//==================================================================================================
//							Beckhoff Automation Poland
//									18.05.2018
//	Struktura interfejsu do obslugi Axis Online
//	v1.1	|| TC v 3.1.4022.16		|| - zmiana nazw struktur 
// 									 ST_FBCoEAX8000SetPositionOffsetIO 	--> ST_FBCoESetPositionOffsetIO
// 									 ST_FBHoldingBrakeCtrlAX8000IO 		--> ST_FBHoldingBrakeCtrlIO
// 									 ST_FBMotorMonitoringAX8000IO 		--> ST_FBMotorMonitoringIO
//  v1.0	|| TC v 3.1.4022.16		|| - pierwsza wersja
//==================================================================================================
TYPE ST_McAxisOnline :
STRUCT
	// Base administration
	mcPower							: ST_MCPowerIO;
	mcStop							: ST_MCStopIO;
	mcHalt							: ST_MCHaltIO;
	mcSS1							: ST_MCStopIO;
	mcSS2							: ST_MCStopIO;
	mcReset							: ST_MCResetIO;
	mcHome							: ST_MCHomeIO;
	mcSetPosition					: ST_MCSetPositionIO;
	stSetPositionOffset				: ST_FBSetPositionOffsetIO;
	// Base move
	mcMoveAbsolute					: ST_MCMoveAbsoluteIO;
	mcMoveRelative					: ST_MCMoveRelativeIO;
	mcMoveVelocity					: ST_MCMoveVelocityIO;
	mcMoveModulo					: ST_MCMoveModuloIO;
	mcMoveAbsolute2					: ST_MCMoveAbsoluteIO;
	mcMoveRelative2					: ST_MCMoveRelativeIO;
	mcMoveVelocity2					: ST_MCMoveVelocityIO;
	mcMoveModulo2					: ST_MCMoveModuloIO;
	mcJog							: ST_MCJogIO;
	// States, parameters, monitoring and diag
	stMotorMonitoring				: ST_FBMotorMonitoringIO;
	stHoldingBrake					: ST_FBHoldingBrakeCtrlIO;
	stNcLimitSwitch					: ST_FBNcSWLimitSwitchCtrlIO;
	stAxisParameter					: Tc2_MC2.ST_AxisParameterSet;
	stDriveRef						: Tc2_EtherCAT.ST_DriveRef;
	stDriveAddress					: Tc2_MC2.ST_DriveAddress;
	stChannelErrorCode				: ST_FBReadChannelErrorCodeIO;
	stStatus						: ST_McAxisStatus;
	// FBs
	stGetDriveRef					: ST_FBGetDriveRefIO;					// IO for FB_GetDriveRef
	mcReadDriveAddress				: ST_MCReadDriveAddressIO;				// IO for MC_ReadDriveAddress
	mcReadParameterSet				: ST_MCReadParameterSetIO;				// IO for MC_ReadParameterSet
	stError							: ST_McAxisOnlineErrorCollection;		// Error collection for all Axis Online functions
	bError							: BOOL;									// General Error flag - all error, FB, NC, drive, communication... check stError for detail
END_STRUCT
END_TYPE

(* stored: Version 1.1.0.1, ProductVersion 3.1.4026.13, FileIdentifier 1040e05450a52b3718c226347e4042459dee8cef, FileSignature 52ca2b1d1d5ce96ca13f1e5682f14ebfa1c234bec118ae1009412476daa953d28524afa8b43aa8278c938f1df601b98e15fb05f85a9c5166142f802fba86411b7b6ab832efc5f74d97a541c4aa92ad2cfeb8e782e95dd72c50c1fa384305956f63551436566b6e0ef09dc17c0ae95bbc38b040a5b1c769aa8f905b04c230f7d0c670c34ebd22352f08ac347581256e981474bc06423b0303cd4300c726c2b9d35dd60b6c8201334fb41ee3a736fd15cb6f8529c07e9dc3dbe396ffe7e563c97105a6d3015225fc6cfb8d7e700387051e8ad6b58c0b45bba83393ca4ab71b5751a374f71dbe1e5f0f913528fd7149203e4d6daf9b84279a81d38e354b91649d57
   DUT ST_McAxisOnline: Id {6ab98389-c989-48b9-b5d8-977bc9b175b3} *)
